(*

.. <legal notes>

legal notes
=================
| SPDX-FileCopyrightText: © 2026 Oleksandr Tiutyk <trofimich@gmail.com>
| SPDX-License-Identifier: LGPL-3.0-only
| For details check: LGPL-3.0-only_

.. _LGPL-3.0-only: https://www.gnu.org/licenses/lgpl-3.0.en.html

.. </legal notes>

*)

TYPE HMI_AUTOMATION_CONTROLLER_BASE_STATUSES :
STRUCT
	Enabled : BOOL;

	HasError : BOOL;
	ErrorMessage : Core.ERROR_MESSAGE;
	ErrorSource : STRING(255);
	ErrorLocalTimestamp : LDATE_AND_TIME;
	ErrorUtcTimestamp : LDATE_AND_TIME;

	OperationalState : OPERATIONAL_STATE;
	OperationalStateName : STRING;
	OperationalStateReason : WSTRING(255);
END_STRUCT
END_TYPE

(* stored: Version 1.1.0.1
   DUT HMI_AUTOMATION_CONTROLLER_BASE_STATUSES: Id {c40c7e9a-c43b-4973-93e1-8c17864d5829} *)
